// TIA Portal V17 export
// export: Created 2024-08-09T12:51:37.7568237Z, ExportSetting WithDefaults, DisplayName Totally Integrated Automation Portal, DisplayVersion V17 Update 7, DisplayName TIA Portal Openness, DisplayVersion V17 Update 7, DisplayName TIA Portal Version Control Interface, DisplayVersion V17, DisplayName STEP 7 Professional, DisplayVersion V17 Update 7, DisplayName STEP 7 Safety, DisplayVersion V17 Update 6, DisplayName WinCC Professional, DisplayVersion V17 Update 7
DATA_BLOCK "DB_Dosage"   // DB38
{ S7_Optimized_Access := 'TRUE' }
VERSION : 0.1
// stored: AutoNumber true, DBAccessibleFromOPCUA true, DBAccessibleFromWebserver true, IsOnlyStoredInLoadMemory false, IsRetainMemResEnabled false, IsWriteProtectedInAS false, MemoryReserve 100
   VAR RETAIN
      TRM_TRANS { S7_SetPoint := 'True'} : Array[0..7] of "S_Tremie_Trans";
      TRM_TRP { S7_SetPoint := 'True'} : Array[0..4] of "S_Tremie_Trappe";
      BP { S7_SetPoint := 'True'} : Array[0..4] of "S_DOSBENNE";
      BR { S7_SetPoint := 'True'} : Array[0..1] of "S_Broyage";
      TRANSF { S7_SetPoint := 'True'} : Array[0..4] of "S_Cir_Trans";
      MLG { S7_SetPoint := 'True'} : Array[0..1] of "S_Melangeuse";
      LIQUIDES_MLG { S7_SetPoint := 'True'} : Array[0..9] of "S_Liquide_Mel";
      VS { S7_SetPoint := 'True'} : Array[0..1] of "S_Verse_Sac";
      DEROUT { S7_SetPoint := 'True'} : "S_Derout_Exp";
      LANC_EXP { S7_SetPoint := 'True'} : "S_Lanc_Exp";
      EXP_DOS { S7_SetPoint := 'True'} : Array[0..1] of "S_Exp_Dos";
   END_VAR
BEGIN
   BR[0..1].EAV_Broy := 1500.0;
END_DATA_BLOCK
